(* PLC project PLC_16099, Beckhoff Automation GmbH TwinCAT PLC Control 3.5.10.30 *)
(* stored: creationDateTime 2018-03-29T14:56:59.9452249, modificationDateTime 2018-03-29T14:56:59.9482329 *)

(* global variable list Frontend *)
{attribute 'Tc2GvlVarNames'}
{attribute 'TcContextName':='PlcTaskStandard'}
(*Diese Liste beinhaltet sämtliche mit dem Frontend ausgetauschten Variablen, plus einige mehr*)
VAR_GLOBAL
	gui_Popup_Nr					:INT;		(*10000er-Stelle bestimmt Typ der Meldung:
												0xxxxx: OK Button
												1xxxxx: OK CANCEL Button
												2xxxxx: YES NO Button
												3xxxxx: YES NO CANCEL Button*)
	gui_Popup_Answer				:INT;		(*0: Bereit
												1: Warten auf Antwort 
												2: Antwort JA (OK)
												3: Antwort NEIN
												4: Antwort CANCEL*)
												
(**************************************************************************************************)
	(*Aktuelle Positionen Achsen, Werte von Sensoren etc.*)
(**************************************************************************************************)
	gui_Play						:BOOL;
	gui_Stop						:BOOL;
	gui_Skipback					:BOOL;
	gui_Skipforward					:BOOL;
	gui_ReqRack						:INT;
	gui_ReqSideTwo					:BOOL;
	gui_ReqSong						:INT;
	gui_ReqNewValuesSong			:BOOL;		(*Frontend verlangt einen neuen Song*)
	gui_Mute						:BOOL;
	gui_IncreaseVolume				:BOOL;
	gui_DecreaseVolume				:BOOL;
	gui_ActRack						:INT;
	gui_SideTwo						:BOOL;
	gui_ActSong						:INT;
	
	(*Noch nicht in XML-Liste*)	
	gui_AktPosMotor1				:REAL;
	gui_AktPosMotor2				:REAL;
	gui_Init						:BOOL;
	gui_Manuellbetrieb				:BOOL;
	gui_RequestOpenDoors			:BOOL;
	gui_Beenden						:BOOL;
END_VAR
